FUNCTION ASSEMBLE_LWORD_FROM_BYTES (* this Function combines the 8 BYTES to a LWORD *)
  (* Standard: 61499-1; Description: Copyright (c) 2026 HR Agrartechnik GmbH This program and the accompanying materials are made available under the terms of the Eclipse Public License 2.0 which is available at https://www.eclipse.org/legal/epl-2.0/ SPDX-License-Identifier: EPL-2.0 *)
  (* Version 1.0, 2026-05-16, Franz Höpfinger, HR Agrartechnik, initial Implementation *)
  PACKAGE eclipse4diac::utils::assembling;
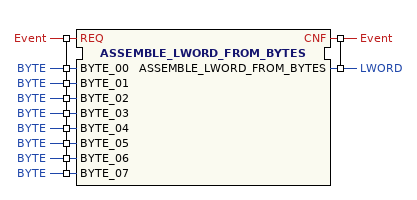
  EVENT_INPUT
    REQ WITH BYTE_00, BYTE_01, BYTE_02, BYTE_03, BYTE_04, BYTE_05, BYTE_06, BYTE_07;
  END_EVENT
  EVENT_OUTPUT
    CNF WITH ASSEMBLE_LWORD_FROM_BYTES;
  END_EVENT
  VAR_INPUT
    BYTE_00 : BYTE;
    BYTE_01 : BYTE;
    BYTE_02 : BYTE;
    BYTE_03 : BYTE;
    BYTE_04 : BYTE;
    BYTE_05 : BYTE;
    BYTE_06 : BYTE;
    BYTE_07 : BYTE;
  END_VAR
  VAR_OUTPUT
    ASSEMBLE_LWORD_FROM_BYTES : LWORD;
  END_VAR
  BODY IN ST:
(* this Function combines the 8 BYTES to a LWORD *)
FUNCTION ASSEMBLE_LWORD_FROM_BYTES : LWORD

VAR_INPUT
	BYTE_00 : BYTE;
	BYTE_01 : BYTE;
	BYTE_02 : BYTE;
	BYTE_03 : BYTE;
	BYTE_04 : BYTE;
	BYTE_05 : BYTE;
	BYTE_06 : BYTE;
	BYTE_07 : BYTE;
END_VAR

ASSEMBLE_LWORD_FROM_BYTES.%B0 := BYTE_00;
ASSEMBLE_LWORD_FROM_BYTES.%B1 := BYTE_01;
ASSEMBLE_LWORD_FROM_BYTES.%B2 := BYTE_02;
ASSEMBLE_LWORD_FROM_BYTES.%B3 := BYTE_03;
ASSEMBLE_LWORD_FROM_BYTES.%B4 := BYTE_04;
ASSEMBLE_LWORD_FROM_BYTES.%B5 := BYTE_05;
ASSEMBLE_LWORD_FROM_BYTES.%B6 := BYTE_06;
ASSEMBLE_LWORD_FROM_BYTES.%B7 := BYTE_07;

END_FUNCTION
  END_BODY
END_FUNCTION
